# EPICS IOC start-up script: iocsh/ethercatmcAnalogInput.iocsh
ethercatmcCreateAsynParam $(MOTOR_PORT) $(ASYNPARAMNAME)      Float64
ethercatmcCreateAsynParam $(MOTOR_PORT) $(ASYNPARAMNAME)_DESC Octet

dbLoadRecords("ethercatmcAnalogInput.template", "P=$(P), R=$(R), MOTOR_PORT=$(MOTOR_PORT), CHNO=$(CHNO), ASYNPARAMNAME=$(ASYNPARAMNAME), PREC=$(PREC), EGU=$(EGU)")
